// TIA Portal V18 export
// export: Created 2025-12-01T12:38:07.3522101Z, ExportSetting None, DisplayName Totally Integrated Automation Portal, DisplayVersion V18 Update 5, DisplayName TIA Portal Openness, DisplayVersion V18 Update 5, DisplayName TIA Portal Teamcenter Gateway, DisplayVersion V18, DisplayName TIA Portal Version Control Interface, DisplayVersion V18, DisplayName STEP 7 Professional, DisplayVersion V18 Update 5, DisplayName STEP 7 Safety, DisplayVersion V18, DisplayName WinCC Professional, DisplayVersion V18 Update 5
DATA_BLOCK "AutoProcessData_Buffer"   // DB1601
{ S7_Optimized_Access := 'FALSE' }
// stored: AutoNumber false
   VAR RETAIN
      DataBuffer : Array[0..55] of "ProcessData";
      DataBuffer_1 : "ProcessData";
      DataBuffer_2 { S7_SetPoint := 'True'} : "ProcessData";
      DataBuffer_3 { S7_SetPoint := 'True'} : "ProcessData";
      DataBuffer_4 { S7_SetPoint := 'True'} : "ProcessData";
      DataBuffer_5 { S7_SetPoint := 'True'} : "ProcessData";
      DataBuffer_6 { S7_SetPoint := 'True'} : "ProcessData";
      VAL { S7_SetPoint := 'True'} : Int;
      SelectButton : Int;
      Button_2 : Bool;
      Button_3 : Bool;
      Button_4 : Bool;
      Button_5 : Bool;
      Button_6 : Bool;
   END_VAR
BEGIN
END_DATA_BLOCK
